(* PLC project Tc2_Utilities.DWORD_TO_OCTSTR Demo, tc3-libraries-kb TwinCAT 3.1 *)
(* stored: creationDateTime 2026-05-10T19:00:00, modificationDateTime 2026-05-10T19:00:00 *)

PROGRAM P_Demo_DWORD_TO_OCTSTR
  VAR
    rResult : T_MaxString;  (* DWORD_TO_OCTSTR 返回值 *)
    bRun : BOOL;  (* 触发一次调用 *)
    v : DWORD;  (* 测试用本地变量 *)
  END_VAR

            // ============================================================
// Tc2_Utilities.DWORD_TO_OCTSTR 演示程序（FUNCTION）
// ============================================================
// 验证步骤：
//   1. 引用 Tc2_Utilities
//   2. 编译 + 登录
//   3. 强制 bRun := TRUE 一个周期
//   4. 在线监视 rResult / 各 demo 变量
// ============================================================

v := 16#FF;
IF bRun THEN
    rResult := DWORD_TO_OCTSTR(v, 8);
    bRun := FALSE;
END_IF;

          
END_PROGRAM
